{attribute 'GeneratedUsingTerminal: EPP1321-0060-0016'}
{attribute addProperty BoxType "EPP1321-0060-0016"}
{attribute addProperty Id "InfoDataAT %I*InfoData_6F19DB2B2"}
{attribute addProperty CRC "532711307"}
{attribute addProperty Size "2"}
TYPE EPP1321_1FC0878B EXTENDS EtcSlaveTerminalBase_947E5A46 :
STRUCT
	{attribute addProperty Name "InfoData"}
	InfoData : InfoData_6F19DB2B;
END_STRUCT
END_TYPE

(* stored: Version 1.2.0.0, ProductVersion 3.1.4024.9
   DUT EPP1321_1FC0878B: Id {a8c6a9d9-a8dc-4e4e-bf13-30eb4d192707} *)
